FUNCTION_BLOCK FB_Pid
VAR
END_VAR

END_FUNCTION_BLOCK

(* stored: Version 1.1.0.1
   POU FB_Pid: Id {4c39227d-65fe-4f51-bba2-df3aff34391c}, SpecialFunc None *)
